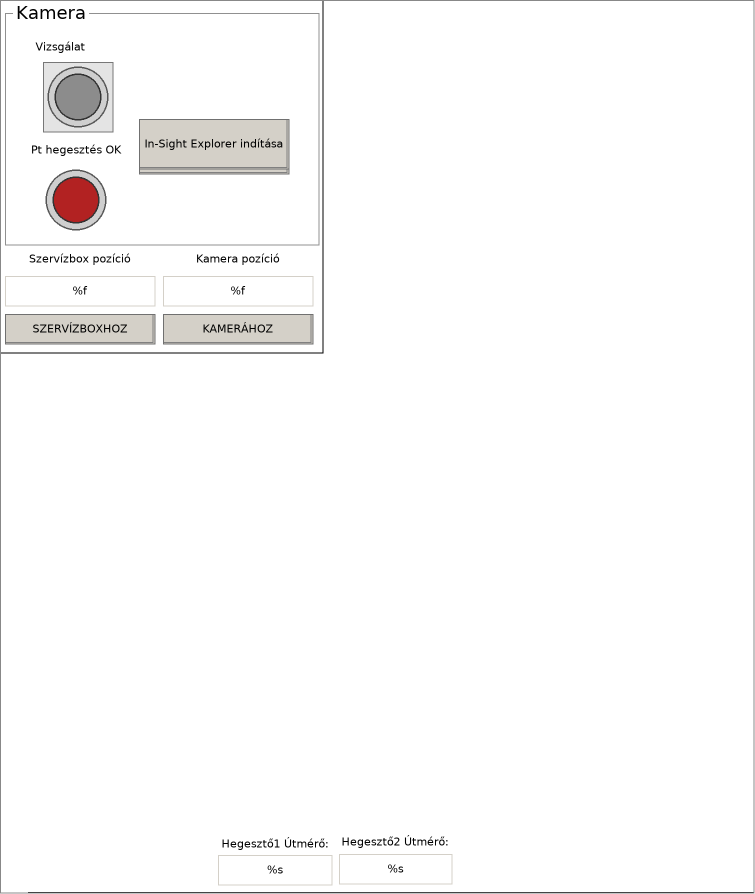
VISUALIZATION Pt1000_oldali_kamera  // 755x894
    Rectangle (0,0 323x353)
    Textfield (218,855 114x30), "%s", text variable: HEGESZTOK.ulHegeszto1Utmero, input disabled if: TRUE
    Label (200,829 150x30), "Hegesztő1 Útmérő:"
    Textfield (339,854 113x30), "%s", text variable: HEGESZTOK.ulHegeszto2Utmero, input disabled if: TRUE
    Label (320,827 150x30), "Hegesztő2 Útmérő:"
    Line (28,892) (753,892)
    GroupBox (5,5 314x240), "Kamera"
        PushSwitch (38,57 70x70), variable: GVL.bPtKameraTrigger, behaviour: TOGGLE, style: Switch-PushSwitch-Gray
        Label (22,32 67x20), "Vizsgálat"
        Button (134,119 150x50), "IV-Navigator indítása", tooltip "A jelölö lézer saját vezérlö szoftvere", pressed state: Laser.bStartFOBADraw
            OnMouseUp: execute { KAMERA.bStartIVNav:=TRUE; }
        Group (18,135 106x95)
            Label (0,0 106x20), "Pt hegesztés OK"
            Lamp1 (18,25 70x70), variable: GVL.bPtKameraHegesztesOK, style: Lamp-Lamp1-Green
            Lamp1 (18,25 70x70), variable: NOT GVL.bPtKameraHegesztesOK, invisible if: GVL.bPtKameraTrigger OR GVL.bPtKameraHegesztesOK, style: Lamp-Lamp1-Red
        Button (134,114 150x50), "In-Sight Explorer indítása", tooltip "A jelölö lézer saját vezérlö szoftvere", pressed state: Laser.bStartFOBADraw
            OnMouseUp: ExecuteCommand ExecuteCommand=ExecuteCommand=[Command=ExecuteClientProgram, Value='C:\Program Files\Cognex\In-Sight\In-Sight Explorer 5.5.0\In-Sight Explorer.exe']
    Textfield (5,276 150x30), "%f", text variable: GVL.lrPtSzervizbox
    Button (5,314 150x30), "SZERVÍZBOXHOZ"
        OnMouseUp: execute { PISTITENGELY.lrPistiPosition:=GVL.lrPtSzervizbox; PISTITENGELY.sPistiAxisCommand:='MOVE'; }
    Label (5,249 150x20), "Szervízbox pozíció"
    Textfield (163,276 150x30), "%f", text variable: GVL.lrPtKameraPosition
        OnMouseClick: write the text variable via VisuDialogs.Numpad, min -10000, max -1
    Button (163,314 150x30), "KAMERÁHOZ"
        OnMouseUp: execute { PISTITENGELY.lrPistiPosition:=GVL.lrPtKameraPosition; PISTITENGELY.sPistiAxisCommand:='MOVE'; }
    Label (163,249 150x20), "Kamera pozíció"
END_VISUALIZATION

(* stored: Version 1.1.0.1, ProductVersion 3.1.4024.11
   Visu Pt1000_oldali_kamera: Id {ce5ceaa2-c4f1-46a7-94df-49584fdf2ebf} *)
